// TIA Portal V17 export
// export: Created 2024-08-09T12:52:50.1221531Z, ExportSetting WithDefaults, DisplayName Totally Integrated Automation Portal, DisplayVersion V17 Update 7, DisplayName TIA Portal Openness, DisplayVersion V17 Update 7, DisplayName TIA Portal Version Control Interface, DisplayVersion V17, DisplayName STEP 7 Professional, DisplayVersion V17 Update 7, DisplayName STEP 7 Safety, DisplayVersion V17 Update 6, DisplayName WinCC Professional, DisplayVersion V17 Update 7
DATA_BLOCK "DB_Lanc_Boucles"   // DB8
VERSION : 0.1
// stored: AutoNumber true, DBAccessibleFromOPCUA true, DBAccessibleFromWebserver true, InstanceOfName Lanc_Boucles, InstanceOfType FB
"Lanc_Boucles"
   // VAR
   //    RAZ_Pt_Zs { ExternalAccessible := 'False'; ExternalVisible := 'False'; ExternalWritable := 'False'} : "S_Suivi_Dosage";
   // END_VAR
BEGIN
END_DATA_BLOCK
